// Mitsubishi GX Works2 project: watch_1   PLC: Q03UDV

PROGRAM MAIN
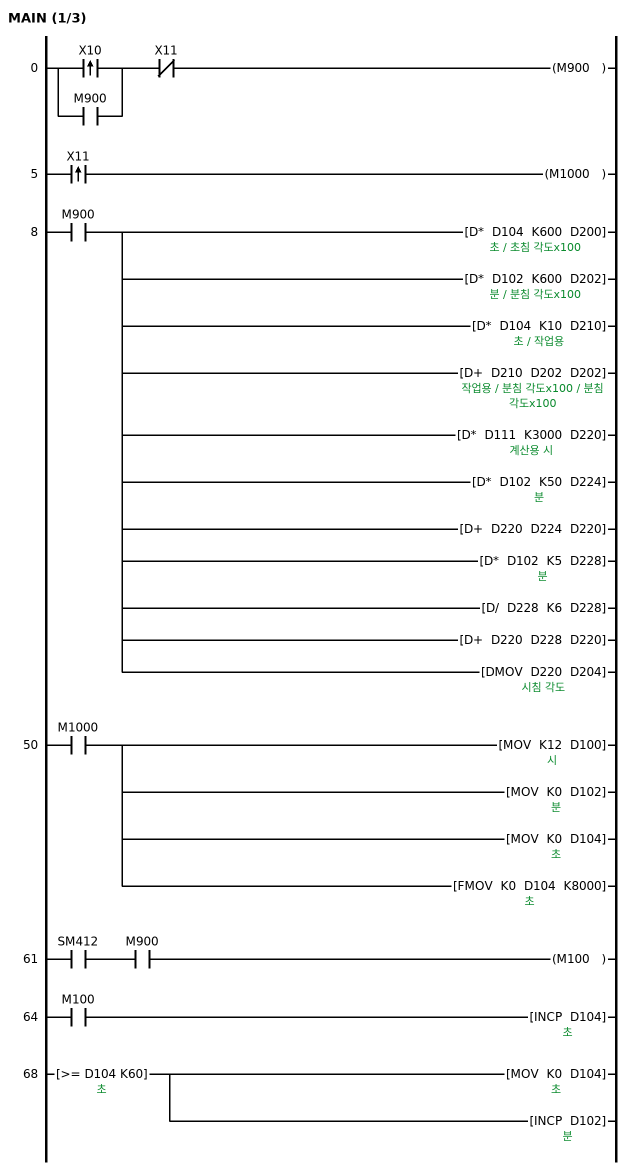
0     LDP     X10
      OR      M900
      ANI     X11
      OUT     M900
5     LDP     X11
      OUT     M1000
8     LD      M900
      D*      D104 K600 D200  ; 초 / 초침 각도x100
      D*      D102 K600 D202  ; 분 / 분침 각도x100
      D*      D104 K10 D210  ; 작업용
      D+      D210 D202 D202
      D*      D111 K3000 D220  ; 계산용 시
      D*      D102 K50 D224
      D+      D220 D224 D220
      D*      D102 K5 D228
      D/      D228 K6 D228
      D+      D220 D228 D220
      DMOV    D220 D204  ; 시침 각도
50    LD      M1000
      MOV     K12 D100  ; 시
      MOV     K0 D102
      MOV     K0 D104
      FMOV    K0 D104 K8000
61    LD      SM412
      AND     M900
      OUT     M100
64    LD      M100
      INCP    D104
68    LD>=    D104 K60  ; 초
      MOV     K0 D104
      INCP    D102
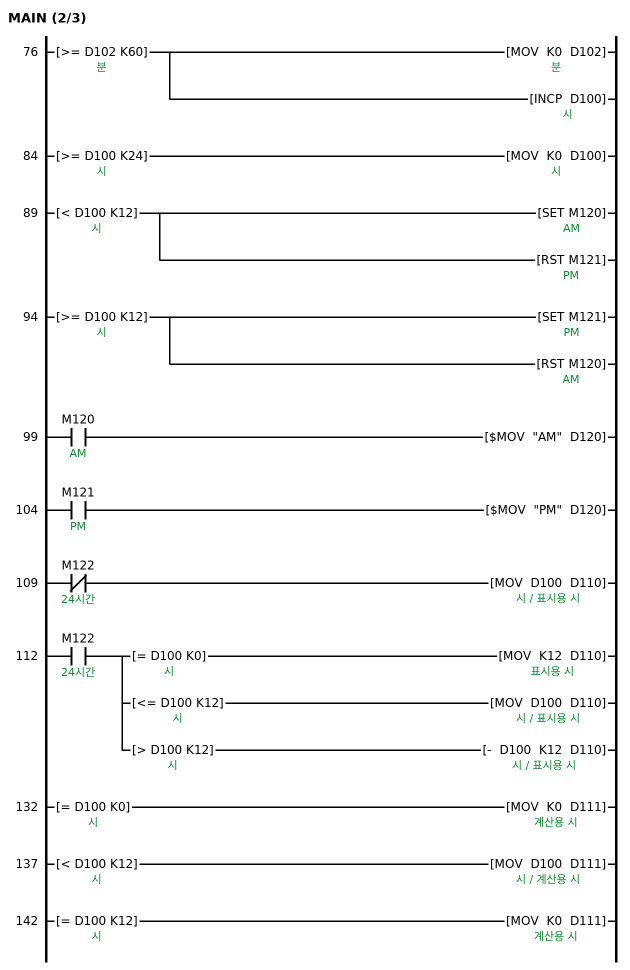
76    LD>=    D102 K60  ; 분
      MOV     K0 D102
      INCP    D100
84    LD>=    D100 K24  ; 시
      MOV     K0 D100
89    LD<     D100 K12  ; 시
      SET     M120  ; AM
      RST     M121  ; PM
94    LD>=    D100 K12  ; 시
      SET     M121  ; PM
      RST     M120  ; AM
99    LD      M120  ; AM
      $MOV    "AM" D120
104   LD      M121  ; PM
      $MOV    "PM" D120
109   LDI     M122  ; 24시간
      MOV     D100 D110  ; 표시용 시
112   LD      M122  ; 24시간
      MPS
      AND=    D100 K0  ; 시
      MOV     K12 D110
      MRD
      AND<=   D100 K12  ; 시
      MOV     D100 D110
      MPP
      AND>    D100 K12  ; 시
      -       D100 K12 D110
132   LD=     D100 K0  ; 시
      MOV     K0 D111
137   LD<     D100 K12  ; 시
      MOV     D100 D111
142   LD=     D100 K12  ; 시
      MOV     K0 D111
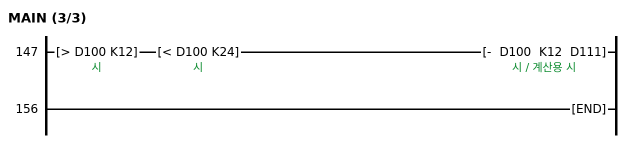
147   LD>     D100 K12  ; 시
      AND<    D100 K24  ; 시
      -       D100 K12 D111
156   END
END_PROGRAM

// device comments not shown above
M123  ; 12시간
D211  ; 작업용
D212  ; 작업용
